ABB RobotStudio station: ESTACION_DEF_ROBOT_20220126-184058.rsstn

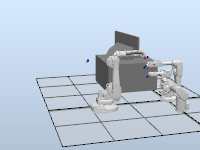
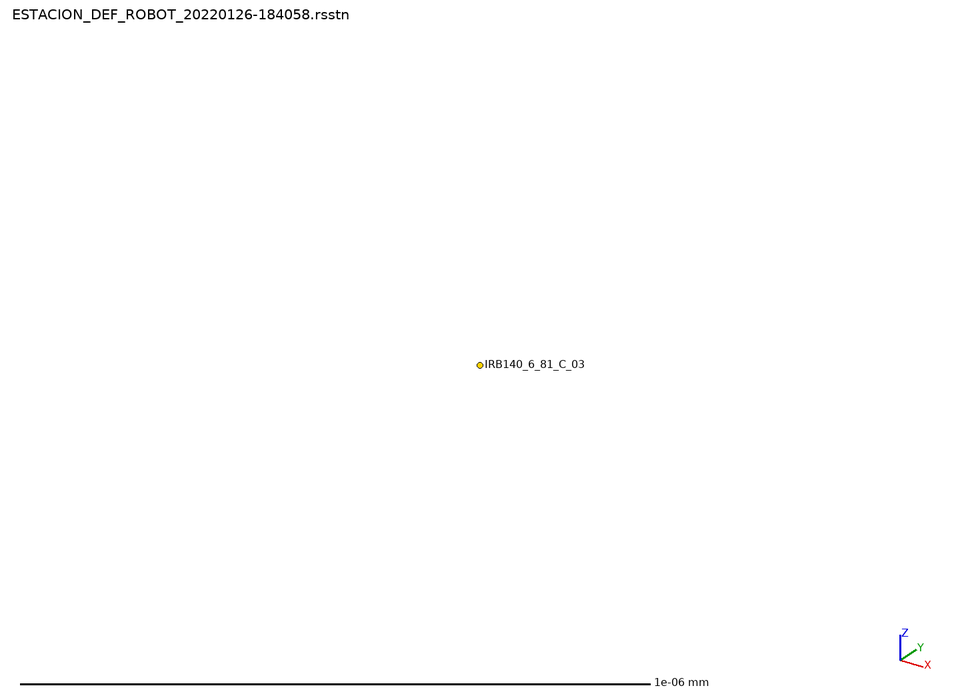
[picture v1: parts stored in the station drawn from their meshes, with robot base, taught points and paths (robot models come from the ABB library and are not in the file)]
Station Station (saved by RobotStudio 21.2.9526.0)
Controller Controlador5
  mechanical unit ROB_1: IRB140_6_81_C_03, 6 joints, base frame (0, 0, 0) mm
Layout (positions relative to the parent item):
  - IRB140_6_81_C_03 [mechanism, from Robots\IRB140_6_81_C_G_03.rslib] at (0, 0, 0) mm; joint values [0, -0.1562, 0.2279, 0, 0.4519, 0] (rad or m)
  - Conjunto_para_piezas_2 [part] at (0, 0, 452.24) mm, rotated rx 90 ry 0 rz 0 deg, size 1400 x 1500 x 1400 mm
  - IRB1660ID_6_155__03 [mechanism, from Robots\IRB1660ID_6_155__03.rslib] at (1658.63, 288.18, 12.54) mm, rotated rx 0 ry 0 rz 180 deg; joint values [0, 0, 0, 0, 0.5236, 0] (rad or m)
  - IRB1300_7_140__01_2 [mechanism, from Robots\IRB1300_7_140__01.rslib] at (0, 779.28, 0) mm; joint values [0, 0, 0, 0, 0.5236, 0] (rad or m)
Targets, tools, work objects and paths stored in the station, written as RAPID:
! task T_ROB1
MODULE Module1
  CONST robtarget Target_10:=[[1714.021,-1416.247,797.687],[1,0,0,0],[0,0,0,0],[9E+09,9E+09,9E+09,9E+09,9E+09,9E+09]];
ENDMODULE

